// This functionblock acts as a stream buffer for use with FB_XmlControl
FUNCTION_BLOCK FB_XmlFileStream EXTENDS FB_StreamBuffer
VAR
    File : FB_FileControl;
  
    BufferInitialised : BOOL := FALSE;
    Buffer : ARRAY [0..(GVL_Param_TcUnit.XUnitBufferSize - 1)] OF BYTE;  
END_VAR

// Appends a string to the buffer
PROPERTY Append : T_MaxString
SET
VAR
    ByteIn : POINTER TO BYTE;
    ByteBuffer : POINTER TO BYTE;
END_VAR
ByteIn := ADR(Append); 
ByteBuffer := _PointerToStringBuffer + _Length; // set start address

REPEAT
  
  WHILE ByteIn^ <> 0 AND _Length < _BufferSize  DO
      ByteBuffer^ := ByteIn^; //Copy the 1st byte
      _Length := _Length + 1; // set new buffer length
      ByteIn := ByteIn + 1; // calculate new start address 
      ByteBuffer := ByteBuffer + 1; // calculate new start address 
  END_WHILE;
  
  IF ByteIn^ <> 0
  THEN
    Flush();
    Clear();
    ByteBuffer := _PointerToStringBuffer;
  END_IF

UNTIL ByteIn^ = 0 END_REPEAT

ByteBuffer := _PointerToStringBuffer + _Length; // String End
ByteBuffer^ := 0; // null terminated string
END_SET
END_PROPERTY

(*
    Deletes the former file (if it exists).
    Opens the file, writes the buffer and closes it.
*)
METHOD CloseFile : SysFile.SysTypes.RTS_IEC_RESULT;
CloseFile := SysDir.CmpErrors.Errors.ERR_OK;
CloseFile := MAX(CloseFile, Flush());
CloseFile := MAX(CloseFile, File.Close());
END_METHOD

(*
    Deletes the former file (if it exists).
    Opens the file, writes the buffer and closes it.
*)
METHOD CreateFile : SysFile.SysTypes.RTS_IEC_RESULT;
CreateFile := SysDir.CmpErrors.Errors.ERR_OK;
CreateFile := MAX(CreateFile, File.Delete(Filename := GVL_Param_TcUnit.xUnitFilePath));
CreateFile := MAX(CreateFile, File.Open(Filename := GVL_Param_TcUnit.xUnitFilePath, FileAccessMode := ACCESS_MODE.AM_WRITE_PLUS));
END_METHOD

//FB_Init is always available implicitly and it is used primarily for initialization.
//The return value is not evaluated. For a specific influence, you can also declare the
//methods explicitly and provide additional code there with the standard initialization
//code. You can evaluate the return value.
METHOD FB_Init: BOOL
VAR_INPUT
    bInitRetains: BOOL; // TRUE: the retain variables are initialized (reset warm / reset cold)
    bInCopyCode: BOOL;  // TRUE: the instance will be copied to the copy code afterward (online change)   
END_VAR
SetBuffer(ADR(Buffer), GVL_Param_TcUnit.XUnitBufferSize);
END_METHOD

(*
    Deletes the former file (if it exists).
    Opens the file, writes the buffer and closes it.
*)
METHOD PRIVATE Flush : SysFile.SysTypes.RTS_IEC_RESULT;
Flush := SysDir.CmpErrors.Errors.ERR_OK;
Flush := MAX(Flush, File.Write(_PointerToStringBuffer, _Length));
Flush := MAX(Flush, File.Close());
Flush := MAX(Flush, File.Open(Filename := GVL_Param_TcUnit.xUnitFilePath, FileAccessMode := ACCESS_MODE.AM_APPEND_PLUS));
END_METHOD

END_FUNCTION_BLOCK

(* stored: Version 1.1.0.1
   POU FB_XmlFileStream: Id {dddd4175-b67a-0902-3b59-1c80dcdfda8c}, SpecialFunc None
   Property Append: Id {3ca21355-e56f-0a40-2994-8442fe8f9a13}
   Set Set: Id {acda1699-b58d-0053-1454-378e0da328d4}
   Method CloseFile: Id {506f243e-65c2-0bad-27d2-c84f4b235bbd}
   Method CreateFile: Id {6244f4a5-e898-0ddb-089d-bad22f5a92db}
   Method FB_init: Id {0874c850-d713-0321-28cd-b342f2f30134}
   Method Flush: Id {d06eec93-628a-0aa6-0431-7060901a9f4e} *)
